{attribute 'linkalways'} 
{attribute 'no_explicit_call' := 'This FB is a CLASS and must be accessed using methods or properties'}
{attribute 'enable_dynamic_creation'}
FUNCTION_BLOCK _ETcVnThresholdType EXTENDS EnumDatatypeBase
VAR
	localData : ETcVnThresholdType;
	activeData : REFERENCE TO ETcVnThresholdType;
	enumBaseDatatype : _DINT(localData);
END_VAR

METHOD PRIVATE AddLocalEnumeration
VAR_INPUT
	Enumeration : T_MAXSTRING;
	Value : ETcVnThresholdType;
END_VAR
AddEnumeration(Enumeration, Value);
END_METHOD

PROPERTY PUBLIC Address : PVOID
GET
Address := ADR(activeData);
END_GET
END_PROPERTY

METHOD PUBLIC ClearReference
VAR_INPUT
END_VAR
activeData REF= localData;
SetBaseDatatypeReference();
END_METHOD

METHOD PUBLIC Clone : I_Datatype
VAR
    pClone : POINTER TO _ETcVnThresholdType;
END_VAR
pClone := __NEW(_ETcVnThresholdType(InitialValue := Value));
Clone := pClone^;
END_METHOD

METHOD FB_init : BOOL
VAR_INPUT
	bInitRetains : BOOL; // if TRUE, the retain variables are initialized (warm start / cold start)
	bInCopyCode : BOOL;  // if TRUE, the instance afterwards gets moved into the copy code (online change)
	InitialValue : ETcVnThresholdType;
END_VAR
localData := InitialValue;
AddBaseDatatype(enumBaseDatatype);
ClearReference();

AddLocalEnumeration('TCVN_TT_BINARY', ETcVnThresholdType.TCVN_TT_BINARY);
AddLocalEnumeration('TCVN_TT_BINARY_INV', ETcVnThresholdType.TCVN_TT_BINARY_INV);
AddLocalEnumeration('TCVN_TT_TRUNC', ETcVnThresholdType.TCVN_TT_TRUNC);
AddLocalEnumeration('TCVN_TT_TOZERO', ETcVnThresholdType.TCVN_TT_TOZERO);
AddLocalEnumeration('TCVN_TT_TOZERO_INV', ETcVnThresholdType.TCVN_TT_TOZERO_INV);
AddLocalEnumeration('TCVN_TT_OTSU_BINARY', ETcVnThresholdType.TCVN_TT_OTSU_BINARY);
AddLocalEnumeration('TCVN_TT_OTSU_BINARY_INV', ETcVnThresholdType.TCVN_TT_OTSU_BINARY_INV);
AddLocalEnumeration('TCVN_TT_OTSU_TRUNC', ETcVnThresholdType.TCVN_TT_OTSU_TRUNC);
AddLocalEnumeration('TCVN_TT_OTSU_TOZERO', ETcVnThresholdType.TCVN_TT_OTSU_TOZERO);
AddLocalEnumeration('TCVN_TT_OTSU_TOZERO_INV', ETcVnThresholdType.TCVN_TT_OTSU_TOZERO_INV);
AddLocalEnumeration('TCVN_TT_TRIANGLE_BINARY', ETcVnThresholdType.TCVN_TT_TRIANGLE_BINARY);
AddLocalEnumeration('TCVN_TT_TRIANGLE_BINARY_INV', ETcVnThresholdType.TCVN_TT_TRIANGLE_BINARY_INV);
AddLocalEnumeration('TCVN_TT_TRIANGLE_TRUNC', ETcVnThresholdType.TCVN_TT_TRIANGLE_TRUNC);
AddLocalEnumeration('TCVN_TT_TRIANGLE_TOZERO', ETcVnThresholdType.TCVN_TT_TRIANGLE_TOZERO);
AddLocalEnumeration('TCVN_TT_TRIANGLE_TOZERO_INV', ETcVnThresholdType.TCVN_TT_TRIANGLE_TOZERO_INV);
END_METHOD

PROPERTY PUBLIC Identifier : T_MAXSTRING
GET
Identifier := 'ETcVnThresholdType';
END_GET
END_PROPERTY

METHOD IsEnumeratorValueEqual : BOOL
VAR_INPUT
	Enumerator : I_KeyValueForwardEnumerator;
END_VAR
VAR
	storedValue : ETcVnThresholdType;
END_VAR
IF NOT Enumerator.TryGet(storedValue) THEN
	RETURN;
END_IF

IsEnumeratorValueEqual := storedValue = activeData;
END_METHOD

METHOD PUBLIC MakeReferenceTo
VAR_INPUT
	ReferenceTarget : REFERENCE TO ETcVnThresholdType;
END_VAR
activeData REF= ReferenceTarget;
SetBaseDatatypeReference();
END_METHOD

METHOD PROTECTED SetBaseDatatypeReference
VAR_INPUT
END_VAR
enumBaseDatatype.MakeReferenceTo(activeData);
END_METHOD

PROPERTY PUBLIC Size : UDINT
GET
Size := SIZEOF(activeData);
END_GET
END_PROPERTY

METHOD TryMakeReferenceTo : BOOL
VAR_INPUT
	Target : I_Datatype;
END_VAR
VAR
	targetAsEnum : I_EnumDatatype;
	pTargetData : POINTER TO ETcVnThresholdType;
END_VAR
IF NOT Target.TryResolveAsEnumDatatype(targetAsEnum) THEN
	RETURN;
END_IF

IF targetAsEnum.Identifier <> Identifier THEN
	RETURN;
END_IF

pTargetData := Target.Address;
activeData REF= pTargetData^;
SetBaseDatatypeReference();
TryMakeReferenceTo := TRUE;
END_METHOD

PROPERTY PUBLIC Value : ETcVnThresholdType
GET
Value := activeData;
END_GET
SET
activeData := Value;
END_SET
END_PROPERTY

END_FUNCTION_BLOCK

(* stored: Version 1.1.0.1, ProductVersion 3.1.4024.12
   POU _ETcVnThresholdType: Id {3c02b2a1-5711-4245-855c-28d089dc75a4}, SpecialFunc None
   Folder Constructor: Id {05c68e85-bc90-41ab-a1a3-a9647d8900c3}
   Folder Private: Id {9c65102f-e144-4440-b23e-864efa59b690}
   Folder Protected: Id {5a4e4a88-7f3c-411a-b931-9e94c159b496}
   Method AddLocalEnumeration: Id {e81fdc11-fd5a-49dc-aa0e-58a9952ad376}
   Property Address: Id {64ed416e-13a7-4ac1-8053-a2c7da87bfbf}
   Get Get: Id {4a43ec49-6ae6-476a-a779-155c3495c1c8}
   Method ClearReference: Id {8cb437cb-983d-43aa-b3a6-837bfd1da693}
   Method Clone: Id {a2661334-fd41-4d1b-b42a-4b1fd2625487}
   Method FB_init: Id {78d0a69d-cd06-47e4-9007-216a8e85ca16}
   Property Identifier: Id {232d988c-82e0-49b4-a335-44bf86145329}
   Get Get: Id {226105f4-d7a0-4415-a06b-96df721e16b2}
   Method IsEnumeratorValueEqual: Id {58f2193b-284e-45b3-a395-e6e7e7b230e9}
   Method MakeReferenceTo: Id {e5682200-c176-4d6c-9cde-b60452b7f925}
   Method SetBaseDatatypeReference: Id {cb57aa3a-f109-49c2-af6f-512c9aa6cdea}
   Property Size: Id {91402fc5-4fcb-4ddc-a904-dc271269cead}
   Get Get: Id {6472788f-42bc-494d-90f9-477be4d30406}
   Method TryMakeReferenceTo: Id {ce974a0c-abd2-4410-84fc-97ff96dbc8ed}
   Property Value: Id {98a0466a-1334-4d20-8592-5936241277e7}
   Get Get: Id {d2f9ecd9-76cd-4093-a137-f4088b4f16ca}
   Set Set: Id {a5f0a2f3-4a1f-4663-99fb-b24c399d0e43} *)
